VAR_GLOBAL
    // M1L0
    Serial_RXBuffer_M1L0 : ComBuffer;
    Serial_TXBuffer_M1L0 : ComBuffer;

    // M2L0
    Serial_RXBuffer_M2L0 : ComBuffer;
    Serial_TXBuffer_M2L0 : ComBuffer;
END_VAR

(* stored: Version 1.1.0.1, ProductVersion 3.1.4022.18
   GVL GVL_COM_Buffers: Id {a8441f26-f9f8-4fbc-842d-41b6657e3ba7} *)
